// TIA Portal project "plc_communication_V17" (V17)

(* hardware
DEVICE "S71500/ET200MP station_1"  S7-1500 station
   slot 0: "Rail_0"  Rack  6ES7 590-1***0-0AA0
   slot 1: "PLC_Remote_Server"  CPU 1511-1 PN  6ES7 511-1AK02-0AB0  V2.8
      slot 3: "CPU display_1"  6ES7591-1AA00-0AA0
      slot 32768: "PROFINET interface_1"  X1
         slot 32769: "Port_1"  X1 P1
         slot 32770: "Port_2"  X1 P2
      slot 34817: "Virtual CP interface port_1"  Virtual CP interface port  Virtual CP interface port
DEVICE "S71500/ET200MP station_2"  S7-1500 station
   slot 0: "Rail_0"  Rack  6ES7 590-1***0-0AA0
   slot 1: "PLC_MAIN_Client"  CPU 1511-1 PN  6ES7 511-1AK02-0AB0  V2.8
      slot 3: "CPU display_1"  6ES7591-1AA00-0AA0
      slot 32768: "PROFINET interface_1"  X1
         slot 32769: "Port_1"  X1 P1
         slot 32770: "Port_2"  X1 P2
      slot 34817: "Virtual CP interface port_1"  Virtual CP interface port  Virtual CP interface port
*)

// ===== PLC "PLC_Remote_Server"  CPU 1511-1 PN =====

VAR_GLOBAL   // PLC tag table "Default tag table"
   "System_Byte" AT %MB1 : Byte;
   "FirstScan" AT %M1.0 : Bool;
   "DiagStatusUpdate" AT %M1.1 : Bool;
   "AlwaysTRUE" AT %M1.2 : Bool;
   "AlwaysFALSE" AT %M1.3 : Bool;
   "Clock_Byte" AT %MB0 : Byte;
   "Clock_10Hz" AT %M0.0 : Bool;
   "Clock_5Hz" AT %M0.1 : Bool;
   "Clock_2.5Hz" AT %M0.2 : Bool;
   "Clock_2Hz" AT %M0.3 : Bool;
   "Clock_1.25Hz" AT %M0.4 : Bool;
   "Clock_1Hz" AT %M0.5 : Bool;
   "Clock_0.625Hz" AT %M0.6 : Bool;
   "Clock_0.5Hz" AT %M0.7 : Bool;
   "Tag_1" AT %M100.0 : Bool;
   "Tag_2" AT %Q0.0 : Bool;
   "Tag_3" AT %I0.0 : Bool;
   "Tag_4" AT %M100.1 : Bool;
   "Tag_5" AT %I1.0 : Bool;
   "Tag_6" AT %Q100.0 : Bool;
   "Tag_7" AT %I100.0 : Bool;
   "Tag_8" AT %I101.0 : Bool;
   "Tag_9" AT %M100.2 : Bool;
   "Tag_10" AT %I101.1 : Bool;
END_VAR

DATA_BLOCK "Server_Config"   // DB2
{ S7_Optimized_Access := 'TRUE' }
VERSION : 0.1
   VAR
      Disconnect : Bool;
      Connect : TCON_IP_v4;
      NDR : Bool;
      DR : Bool;
      Error : Bool;
      Status : Word;
   END_VAR
BEGIN
   Connect.InterfaceId := 64;
   Connect.ConnectionType := 11;
   Connect.ActiveEstablished := 0;
   Connect.RemoteAddress.ADDR[1] := 0;
   Connect.RemoteAddress.ADDR[2] := 0;
   Connect.RemoteAddress.ADDR[3] := 0;
   Connect.RemoteAddress.ADDR[4] := 0;
   Connect.RemotePort := 0;
   Connect.ID := 1;
   Connect.LocalPort := 502;
END_DATA_BLOCK

DATA_BLOCK "Server_Data"   // DB3
{ S7_Optimized_Access := 'FALSE' }
VERSION : 0.1
   VAR
      "Send _Data" : Array[0..15] of Word;
   END_VAR
BEGIN
END_DATA_BLOCK

DATA_BLOCK "GET/PUT DATA"   // DB4
{ S7_Optimized_Access := 'FALSE' }
VERSION : 0.1
   VAR
      GET : Struct
         "GET SEND DATA" : Array[0..3] of Word;
      END_STRUCT;
      PUT : Struct
         "PUT RECIEVED DATA" : Array[0..3] of Word;
      END_STRUCT;
   END_VAR
BEGIN
END_DATA_BLOCK

ORGANIZATION_BLOCK "Main_Remote_Server"   // OB1, LAD, ProgramCycle
TITLE = "Main Program Sweep (Cycle)"
{ S7_Optimized_Access := 'TRUE' }
VERSION : 0.1
   VAR_INPUT
      Initial_Call : Bool;   // Initial call of this OB
      Remanence : Bool;   // =True, if remanent data are available
   END_VAR
BEGIN

REGION Network 1
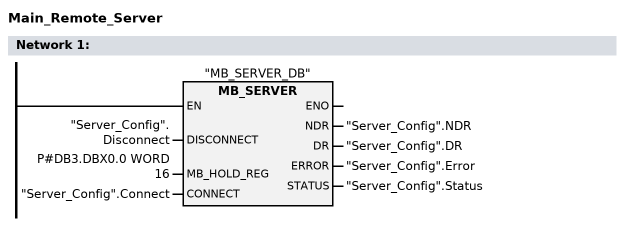
   "MB_SERVER_DB"(DISCONNECT := "Server_Config".Disconnect,   // MB_SERVER
                  MB_HOLD_REG := P#DB3.DBX0.0 WORD 16,
                  CONNECT := "Server_Config".Connect,
                  NDR => "Server_Config".NDR,
                  DR => "Server_Config".DR,
                  ERROR => "Server_Config".Error,
                  STATUS => "Server_Config".Status);
END_REGION
END_ORGANIZATION_BLOCK

// ===== PLC "PLC_MAIN_Client"  CPU 1511-1 PN =====

VAR_GLOBAL   // PLC tag table "Default tag table"
   "System_Byte" AT %MB1 : Byte;
   "FirstScan" AT %M1.0 : Bool;
   "DiagStatusUpdate" AT %M1.1 : Bool;
   "AlwaysTRUE" AT %M1.2 : Bool;
   "AlwaysFALSE" AT %M1.3 : Bool;
   "Clock_Byte" AT %MB0 : Byte;
   "Clock_10Hz" AT %M0.0 : Bool;
   "Clock_5Hz" AT %M0.1 : Bool;
   "Clock_2.5Hz" AT %M0.2 : Bool;
   "Clock_2Hz" AT %M0.3 : Bool;
   "Clock_1.25Hz" AT %M0.4 : Bool;
   "Clock_1Hz" AT %M0.5 : Bool;
   "Clock_0.625Hz" AT %M0.6 : Bool;
   "Clock_0.5Hz" AT %M0.7 : Bool;
END_VAR

DATA_BLOCK "Modbus_Config"   // DB2
{ S7_Optimized_Access := 'TRUE' }
VERSION : 0.1
   VAR
      Disconnect : Bool;
      MB_MODE : USInt;
      MB_DATA_ADDR : UDInt := 40001;
      MB_DATA_LEN : USInt;
      connect : TCON_IP_v4;
      done : Bool;
      busy : Bool;
      error : Bool;
      status : Word;
   END_VAR
BEGIN
   connect.ConnectionType := 11;
   connect.ID := 2;
   connect.ActiveEstablished := 1;
   connect.RemotePort := 502;
   connect.RemoteAddress.ADDR[1] := 192;
   connect.RemoteAddress.ADDR[2] := 168;
   connect.RemoteAddress.ADDR[3] := 0;
   connect.RemoteAddress.ADDR[4] := 3;
   connect.InterfaceId := 64;
END_DATA_BLOCK

DATA_BLOCK "Modbus_Data"   // DB3
{ S7_Optimized_Access := 'FALSE' }
VERSION : 0.1
   VAR
      data : Array[0..15] of Word;
   END_VAR
BEGIN
END_DATA_BLOCK

DATA_BLOCK "GET_config"   // DB6
{ S7_Optimized_Access := 'FALSE' }
VERSION : 0.1
   VAR
      GET : Struct
         NDR : Bool;
         ERROR : Bool;
         STATUS : Word;
         "GET READ DATA" : Array[0..3] of Word;
      END_STRUCT;
      PUT : Struct
         DONE : Bool;
         ERROR : Bool;
         STATUS : Word;
         "PUT SEND DATA" : Array[0..3] of Word;
      END_STRUCT;
   END_VAR
BEGIN
END_DATA_BLOCK

// folder: System blocks/Program resources

DATA_BLOCK "IEC_Counter_0_DB"   // DB4
{ S7_Optimized_Access := 'TRUE' }
AUTHOR : Simatic
FAMILY : IEC
NAME : CNTR
VERSION : 1.0
// stored: InstanceOfName IEC_COUNTER
"IEC_COUNTER"
BEGIN
END_DATA_BLOCK

// folder: (top level)

ORGANIZATION_BLOCK "Main_Master_Client"   // OB1, LAD, ProgramCycle
TITLE = "Main Program Sweep (Cycle)"
{ S7_Optimized_Access := 'TRUE' }
VERSION : 0.1
   VAR_INPUT
      Initial_Call : Bool;   // Initial call of this OB
      Remanence : Bool;   // =True, if remanent data are available
   END_VAR
BEGIN

REGION Network 1
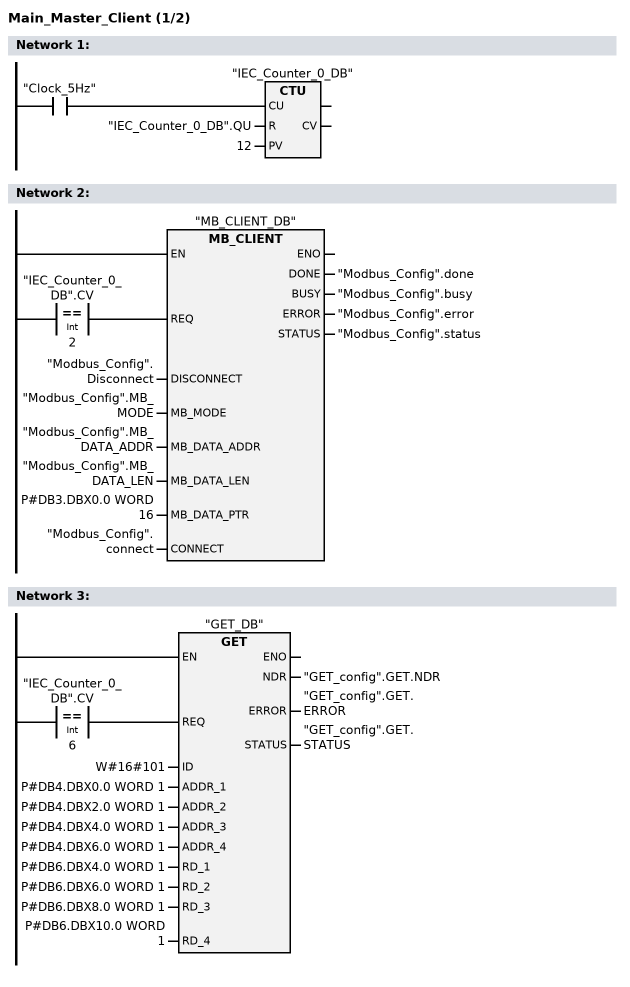
   "IEC_Counter_0_DB".CTU(CU := "Clock_5Hz", R := "IEC_Counter_0_DB".QU, PV := 12);
END_REGION

REGION Network 2
   "MB_CLIENT_DB"(REQ := "IEC_Counter_0_DB".CV = 2,   // MB_CLIENT
                  DISCONNECT := "Modbus_Config".Disconnect,
                  MB_MODE := "Modbus_Config".MB_MODE,
                  MB_DATA_ADDR := "Modbus_Config".MB_DATA_ADDR,
                  MB_DATA_LEN := "Modbus_Config".MB_DATA_LEN,
                  MB_DATA_PTR := P#DB3.DBX0.0 WORD 16,
                  CONNECT := "Modbus_Config".connect,
                  DONE => "Modbus_Config".done,
                  BUSY => "Modbus_Config".busy,
                  ERROR => "Modbus_Config".error,
                  STATUS => "Modbus_Config".status);
END_REGION

REGION Network 3
   "GET_DB"(REQ := "IEC_Counter_0_DB".CV = 6,   // GET
            ID := W#16#101,
            ADDR_1 := P#DB4.DBX0.0 WORD 1,
            ADDR_2 := P#DB4.DBX2.0 WORD 1,
            ADDR_3 := P#DB4.DBX4.0 WORD 1,
            ADDR_4 := P#DB4.DBX6.0 WORD 1,
            RD_1 := P#DB6.DBX4.0 WORD 1,
            RD_2 := P#DB6.DBX6.0 WORD 1,
            RD_3 := P#DB6.DBX8.0 WORD 1,
            RD_4 := P#DB6.DBX10.0 WORD 1,
            NDR => "GET_config".GET.NDR,
            ERROR => "GET_config".GET.ERROR,
            STATUS => "GET_config".GET.STATUS);
END_REGION

REGION Network 4
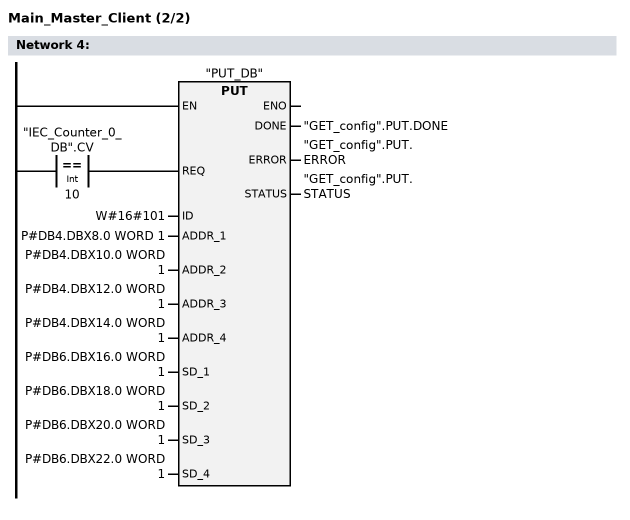
   "PUT_DB"(REQ := "IEC_Counter_0_DB".CV = 10,   // PUT
            ID := W#16#101,
            ADDR_1 := P#DB4.DBX8.0 WORD 1,
            ADDR_2 := P#DB4.DBX10.0 WORD 1,
            ADDR_3 := P#DB4.DBX12.0 WORD 1,
            ADDR_4 := P#DB4.DBX14.0 WORD 1,
            SD_1 := P#DB6.DBX16.0 WORD 1,
            SD_2 := P#DB6.DBX18.0 WORD 1,
            SD_3 := P#DB6.DBX20.0 WORD 1,
            SD_4 := P#DB6.DBX22.0 WORD 1,
            DONE => "GET_config".PUT.DONE,
            ERROR => "GET_config".PUT.ERROR,
            STATUS => "GET_config".PUT.STATUS);
END_REGION
END_ORGANIZATION_BLOCK